// TIA Portal V17 export
// export: Created 2021-12-03T08:13:08.04302Z, ExportSetting WithDefaults, DisplayName Totally Integrated Automation Portal, DisplayVersion V17, DisplayName TIA Portal Openness, DisplayVersion V17, DisplayName TIA Portal Version Control Interface, DisplayVersion V17, DisplayName STEP 7 Professional, DisplayVersion V17, DisplayName STEP 7 Safety, DisplayVersion V17, DisplayName WinCC Advanced, DisplayVersion V17
FUNCTION "FC_Signalization" : Void   // FC801, FBD
VERSION : 0.1
// stored: AutoNumber false, IsIECCheckEnabled false, UDAEnableTagReadback false
BEGIN

REGION Network 2: Пульт P1 Ack
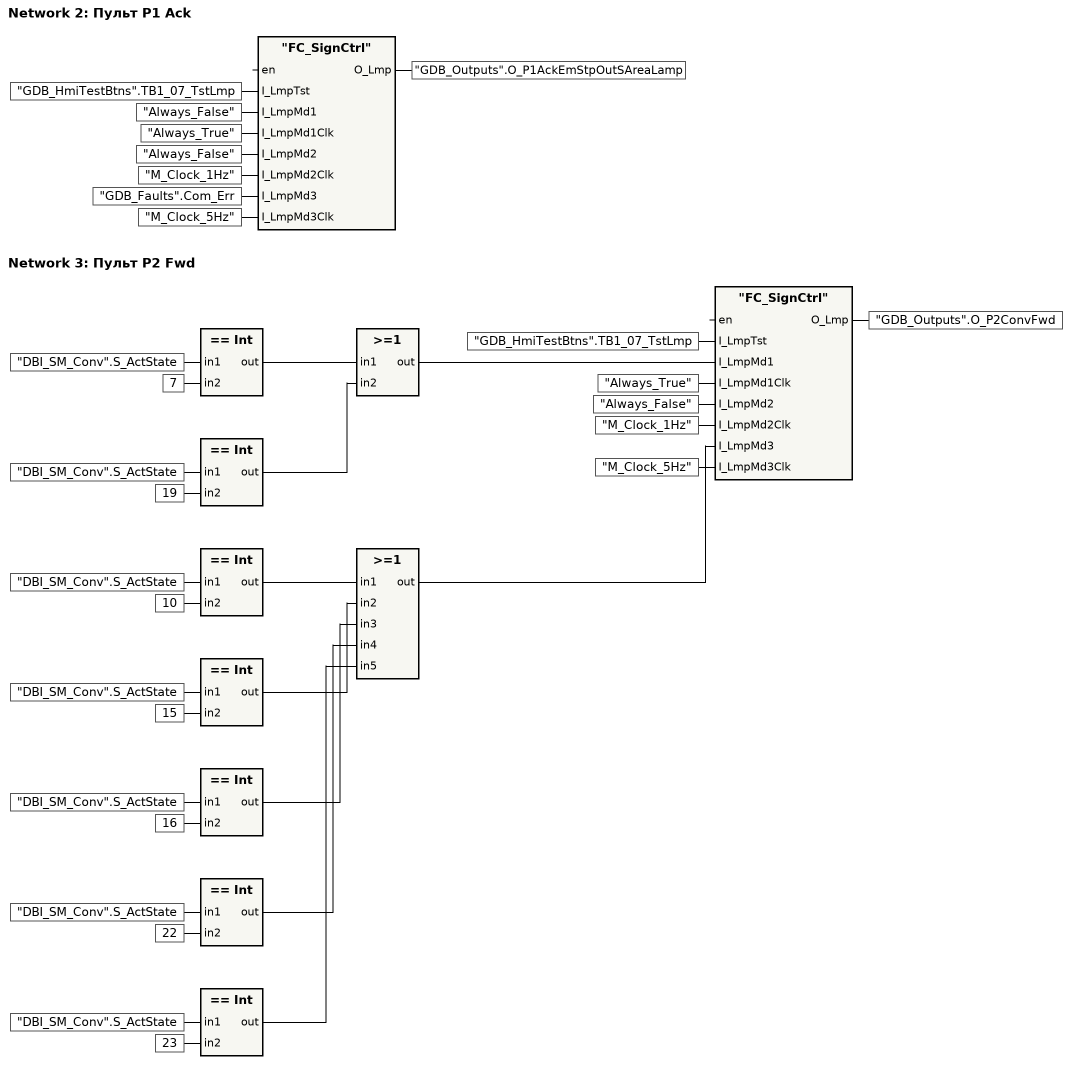
   "FC_SignCtrl"(I_LmpTst := "GDB_HmiTestBtns".TB1_07_TstLmp,
                 I_LmpMd1 := "Always_False",
                 I_LmpMd1Clk := "Always_True",
                 I_LmpMd2 := "Always_False",
                 I_LmpMd2Clk := "M_Clock_1Hz",
                 I_LmpMd3 := "GDB_Faults".Com_Err,
                 I_LmpMd3Clk := "M_Clock_5Hz",
                 O_Lmp => "GDB_Outputs".O_P1AckEmStpOutSAreaLamp);
END_REGION

REGION Network 3: Пульт P2 Fwd
   "FC_SignCtrl"(I_LmpTst := "GDB_HmiTestBtns".TB1_07_TstLmp,
                 I_LmpMd1 := ("DBI_SM_Conv".S_ActState = 7) OR ("DBI_SM_Conv".S_ActState = 19),
                 I_LmpMd1Clk := "Always_True",
                 I_LmpMd2 := "Always_False",
                 I_LmpMd2Clk := "M_Clock_1Hz",
                 I_LmpMd3 := ("DBI_SM_Conv".S_ActState = 10) OR ("DBI_SM_Conv".S_ActState = 15) OR ("DBI_SM_Conv".S_ActState = 16) OR ("DBI_SM_Conv".S_ActState = 22) OR ("DBI_SM_Conv".S_ActState = 23),
                 I_LmpMd3Clk := "M_Clock_5Hz",
                 O_Lmp => "GDB_Outputs".O_P2ConvFwd);
END_REGION

REGION Network 4: Пульт P2 Bwd
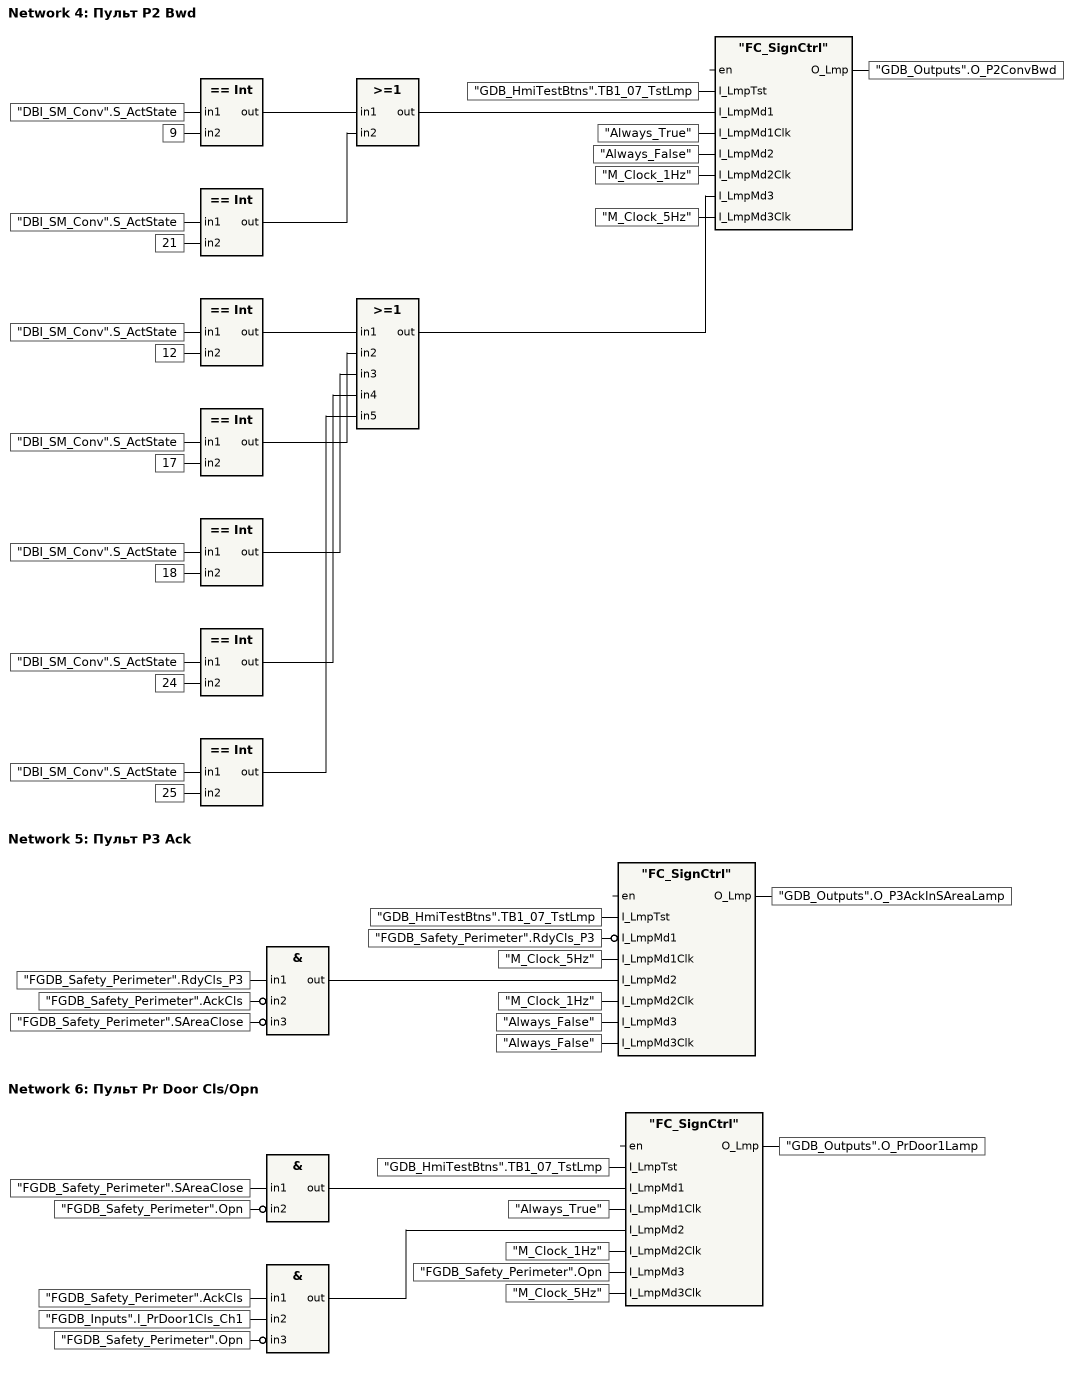
   "FC_SignCtrl"(I_LmpTst := "GDB_HmiTestBtns".TB1_07_TstLmp,
                 I_LmpMd1 := ("DBI_SM_Conv".S_ActState = 9) OR ("DBI_SM_Conv".S_ActState = 21),
                 I_LmpMd1Clk := "Always_True",
                 I_LmpMd2 := "Always_False",
                 I_LmpMd2Clk := "M_Clock_1Hz",
                 I_LmpMd3 := ("DBI_SM_Conv".S_ActState = 12) OR ("DBI_SM_Conv".S_ActState = 17) OR ("DBI_SM_Conv".S_ActState = 18) OR ("DBI_SM_Conv".S_ActState = 24) OR ("DBI_SM_Conv".S_ActState = 25),
                 I_LmpMd3Clk := "M_Clock_5Hz",
                 O_Lmp => "GDB_Outputs".O_P2ConvBwd);
END_REGION

REGION Network 5: Пульт P3 Ack
   "FC_SignCtrl"(I_LmpTst := "GDB_HmiTestBtns".TB1_07_TstLmp,
                 I_LmpMd1 := NOT "FGDB_Safety_Perimeter".RdyCls_P3,
                 I_LmpMd1Clk := "M_Clock_5Hz",
                 I_LmpMd2 := "FGDB_Safety_Perimeter".RdyCls_P3 AND NOT "FGDB_Safety_Perimeter".AckCls AND NOT "FGDB_Safety_Perimeter".SAreaClose,
                 I_LmpMd2Clk := "M_Clock_1Hz",
                 I_LmpMd3 := "Always_False",
                 I_LmpMd3Clk := "Always_False",
                 O_Lmp => "GDB_Outputs".O_P3AckInSAreaLamp);
END_REGION

REGION Network 6: Пульт Pr Door Cls/Opn
   "FC_SignCtrl"(I_LmpTst := "GDB_HmiTestBtns".TB1_07_TstLmp,
                 I_LmpMd1 := "FGDB_Safety_Perimeter".SAreaClose AND NOT "FGDB_Safety_Perimeter".Opn,
                 I_LmpMd1Clk := "Always_True",
                 I_LmpMd2 := "FGDB_Safety_Perimeter".AckCls AND "FGDB_Inputs".I_PrDoor1Cls_Ch1 AND NOT "FGDB_Safety_Perimeter".Opn,
                 I_LmpMd2Clk := "M_Clock_1Hz",
                 I_LmpMd3 := "FGDB_Safety_Perimeter".Opn,
                 I_LmpMd3Clk := "M_Clock_5Hz",
                 O_Lmp => "GDB_Outputs".O_PrDoor1Lamp);
END_REGION

REGION Network 7: Состояние Красный
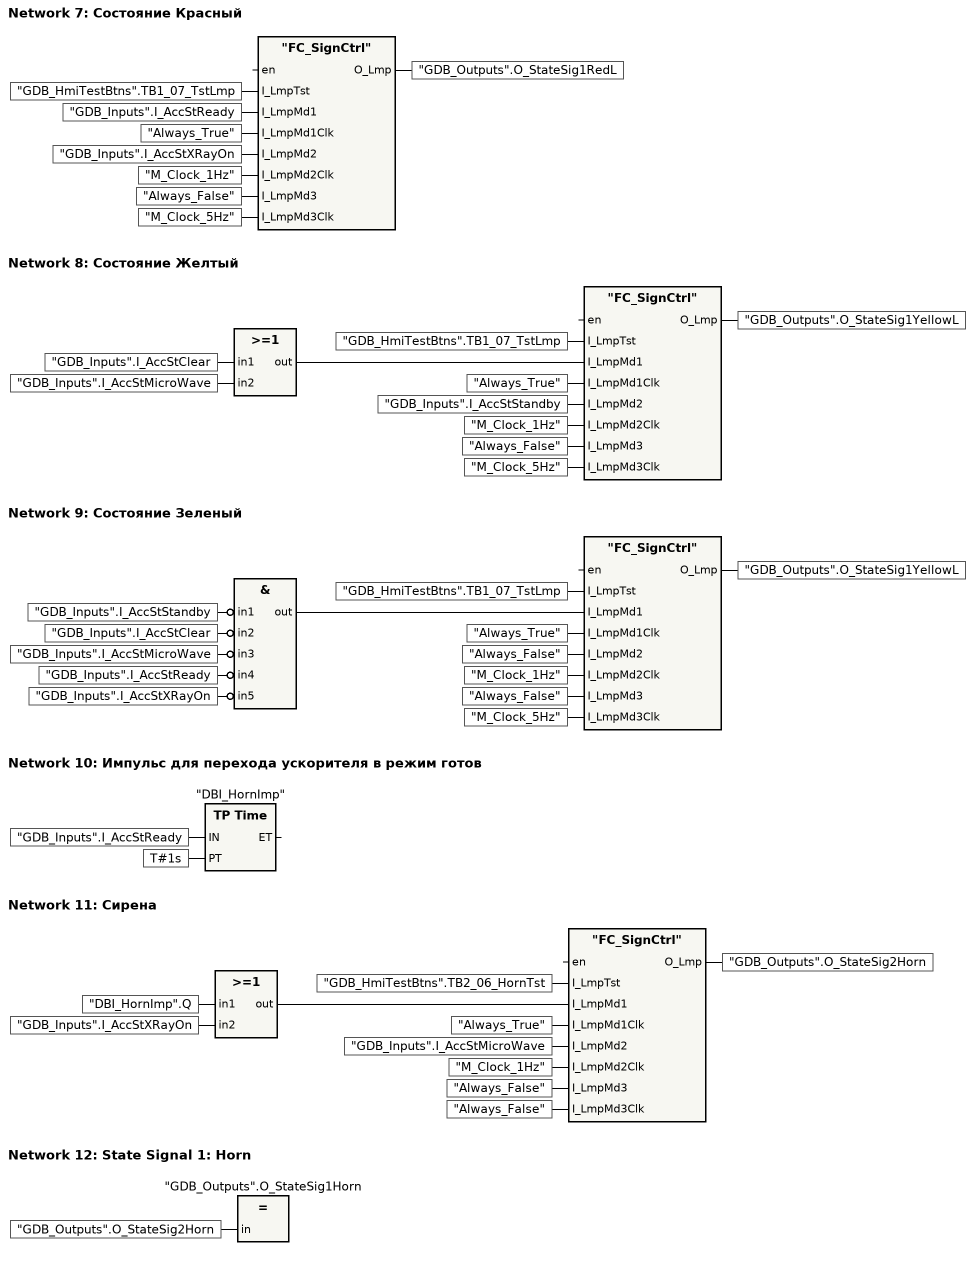
   "FC_SignCtrl"(I_LmpTst := "GDB_HmiTestBtns".TB1_07_TstLmp,
                 I_LmpMd1 := "GDB_Inputs".I_AccStReady,
                 I_LmpMd1Clk := "Always_True",
                 I_LmpMd2 := "GDB_Inputs".I_AccStXRayOn,
                 I_LmpMd2Clk := "M_Clock_1Hz",
                 I_LmpMd3 := "Always_False",
                 I_LmpMd3Clk := "M_Clock_5Hz",
                 O_Lmp => "GDB_Outputs".O_StateSig1RedL);
END_REGION

REGION Network 8: Состояние Желтый
   "FC_SignCtrl"(I_LmpTst := "GDB_HmiTestBtns".TB1_07_TstLmp,
                 I_LmpMd1 := "GDB_Inputs".I_AccStClear OR "GDB_Inputs".I_AccStMicroWave,
                 I_LmpMd1Clk := "Always_True",
                 I_LmpMd2 := "GDB_Inputs".I_AccStStandby,
                 I_LmpMd2Clk := "M_Clock_1Hz",
                 I_LmpMd3 := "Always_False",
                 I_LmpMd3Clk := "M_Clock_5Hz",
                 O_Lmp => "GDB_Outputs".O_StateSig1YellowL);
END_REGION

REGION Network 9: Состояние Зеленый
   "FC_SignCtrl"(I_LmpTst := "GDB_HmiTestBtns".TB1_07_TstLmp,
                 I_LmpMd1 := NOT "GDB_Inputs".I_AccStStandby AND NOT "GDB_Inputs".I_AccStClear AND NOT "GDB_Inputs".I_AccStMicroWave AND NOT "GDB_Inputs".I_AccStReady AND NOT "GDB_Inputs".I_AccStXRayOn,
                 I_LmpMd1Clk := "Always_True",
                 I_LmpMd2 := "Always_False",
                 I_LmpMd2Clk := "M_Clock_1Hz",
                 I_LmpMd3 := "Always_False",
                 I_LmpMd3Clk := "M_Clock_5Hz",
                 O_Lmp => "GDB_Outputs".O_StateSig1YellowL);
END_REGION

REGION Network 10: Импульс для перехода ускорителя в режим готов
   "DBI_HornImp".TP(IN := "GDB_Inputs".I_AccStReady, PT := T#1s);
END_REGION

REGION Network 11: Сирена
   "FC_SignCtrl"(I_LmpTst := "GDB_HmiTestBtns".TB2_06_HornTst,
                 I_LmpMd1 := "DBI_HornImp".Q OR "GDB_Inputs".I_AccStXRayOn,
                 I_LmpMd1Clk := "Always_True",
                 I_LmpMd2 := "GDB_Inputs".I_AccStMicroWave,
                 I_LmpMd2Clk := "M_Clock_1Hz",
                 I_LmpMd3 := "Always_False",
                 I_LmpMd3Clk := "Always_False",
                 O_Lmp => "GDB_Outputs".O_StateSig2Horn);
END_REGION

REGION Network 12: State Signal 1: Horn
   "GDB_Outputs".O_StateSig1Horn := "GDB_Outputs".O_StateSig2Horn;
END_REGION
END_FUNCTION
